// Brief: setup Arm Cart Control
FUNCTION_BLOCK PUBLIC FB_SetupCtrlCart EXTENDS FB_SetupArmCtrlBase
VAR_INPUT
END_VAR
VAR_OUTPUT
END_VAR
VAR
END_VAR

END_FUNCTION_BLOCK

(* stored: Version 1.1.0.1, ProductVersion 3.1.4024.12
   POU FB_SetupCtrlCart: Id {4fa06658-3c16-4ac9-904b-65722ac0872f}, SpecialFunc None *)
